// TwinCAT 3 PLC project Sample
// ProgramVersion: 3.1.4024.0
// libraries:
//   Tc2_Standard, * (Beckhoff Automation GmbH)
//   Tc2_System, * (Beckhoff Automation GmbH)
//   Tc3_Module, * (Beckhoff Automation GmbH)
// project tree:
//   GVLs/ Deskval.TcGVL
//   / PlcTask.TcTTO
//   POUs/ MAIN.TcPOU
// real-time tasks:
//   TASK PlcTask: cycle T#10ms, priority 20, ADS port 350

CONFIGURATION Sample
    RESOURCE PLC ON TwinCAT3
        TASK PlcTask(INTERVAL := T#10ms, PRIORITY := 20);
        PROGRAM MAIN WITH PlcTask : MAIN;
    END_RESOURCE
END_CONFIGURATION

// ---- GVLs/Deskval.TcGVL
{attribute 'qualified_only'}
VAR_GLOBAL
	
	(*
	─────────────────────────────────────────────────────────────────────────────────────────────
	CAUTION:
	─────────────────────────────────────────────────────────────────────────────────────────────
		Deskval Workbench is preconfigured to work with this Global Variable List 
		Do not change neither name of this Global Variable List nor its content in any way.		 
	───────────────────────────────────────────────────────────────────────────────────────────── 
	*)
	
	AdsTagsFromDeskval_Boolean 	:	ARRAY[0..127] OF BOOL;			// Written by Deskval Workbench.
	AdsTagsFromDeskval_Double 	:	ARRAY[0..63] OF LREAL;			// Written by Deskval Workbench.
	AdsTagsFromDeskval_String 	:	ARRAY[0..31] OF STRING(255);	// Written by Deskval Workbench.
	AdsTagsToDeskval_Boolean 	:	ARRAY[0..127] OF BOOL;			// Read by Deskval Workbench.
	AdsTagsToDeskval_Double 	:	ARRAY[0..63] OF LREAL;			// Read by Deskval Workbench.
	AdsTagsToDeskval_String 	:	ARRAY[0..31] OF STRING(255);	// Read by Deskval Workbench.
	BatchTags 					:	ARRAY[0..31] OF STRING(255);	// Read/Write by Deskval Workbench.
	
END_VAR

// ---- POUs/MAIN.TcPOU
PROGRAM MAIN
VAR
	myTimer					: TON;
	randomNumberGenerator	: DRAND();
	randomNumber			: LREAL;
	count					: WORD;
END_VAR

(*
	■ What is exchanged between Twincat Plc and Deskval Workbench ?  							
						Deskval Workbech exchanges its built-in AdsTags in a directional manner. 
						Deskval Workbench exchanges its built-in BatchTags, in a Readonly manner.	
	■ What is required in the Plc project ?
			Twincat Plc Project should have a Global Variable List, named as Deskval with a specific content. It is provided in this project.
					
						
	■ AdsTags				┌───────────────────────────────────────────────────────────────┐		┌───────────────────────────┐
							│ 						Twincat Plc Project         			│		│ 	  Deskval Workbench 	│    
							├───────────────────────────────────────────────────────────────┤		├───────────────────────────┤
							│															 	│		│         Ads Tags   		│     
							│															 	│		│							│                    
			┌────────────── │ 	AdsTagsFromDeskval_Boolean		AdsTagsToDeskval_Boolean	│ ────	► 128 Boolean	128 Boolean ►  ──────────────┐
			│	┌────────── │ 	AdsTagsFromDeskval_Double		AdsTagsToDeskval_Double		│ ────	► 64 Double		64 Double  	►  ──────────┐	 │
			│	│	┌──────	│ 	AdsTagsFromDeskval_String		AdsTagsToDeskval_String		│ ────	► 32 String    	32 String	►  ──────┐	 │	 │
			│	│	│		└───────────────────────────────────────────────────────────────┘		└───────────────────────────┘		 │	 │	 │
			│	│	└────────────────────────────────────────────────────────────────────────────────────────────────────────────────────┘	 │	 │
			│	└────────────────────────────────────────────────────────────────────────────────────────────────────────────────────────────┘	 │
			└────────────────────────────────────────────────────────────────────────────────────────────────────────────────────────────────────┘	

	■ BatchTags				┌───────────────────────────────────────────────────────────────┐		┌───────────────────────────┐
							│ 						Twincat Plc Project         			│		│ 	  Deskval Workbench* 	│    
							├───────────────────────────────────────────────────────────────┤		├───────────────────────────┤
							│															 	│		│       Batch Tags  		│     
							│							BatchTags							│ ◄───►	│		 32 String			│    
							└───────────────────────────────────────────────────────────────┘		└───────────────────────────┘			
			¹ If a Deskval BatchTag is configured to get its value from Ads, then Deskval will Read it from the Plc

	────────────────────────────────────────────────────────────────────────────────────────────────────
	Description : This is a Sample Plc Program to demonstrate Ads Communication with Deskval Workbench.
	──────────────────────────────────────────────────────────────────────────────────────────────────── *)
myTimer(IN:=TRUE, PT:=T#1S);

// On Timer Tick
IF(myTimer.Q) THEN
	
	//Get a Random Number
	randomNumberGenerator(Seed:=17, Num=>randomNumber);		
	
	// Write to First Boolean Tag
	Deskval.AdsTagsToDeskval_Boolean[0] := NOT(Deskval.AdsTagsToDeskval_Boolean[0]);
	
	// Write to Second Num Tag
	Deskval.AdsTagsToDeskval_Double[1] 	:= randomNumber*100;
	
	// Write to Third String Tag
	Deskval.AdsTagsToDeskval_String[2] 	:= CONCAT('Count ',WORD_TO_STRING(count));
	
	// Write To Fourth Batch Tag
	Deskval.BatchTags[3] 				:= CONCAT('Some Batch ',WORD_TO_STRING(count));
	
	// Reset Timer
	myTimer(IN:=FALSE);

	//Increment count
	count := count + 1;
END_IF

END_PROGRAM
